(* IEC 61131-3 sources: POC_HINCAPIE/Project/SIEMENS/DIGSI/Guadalupe/TMP/CFC/7344242.46252 (part 2) *)

     (* 0133 - GDL69TRF2F003_.Application.FG1_UserDef.FB2_Universal.SPS6 *)
     EXV_SPS_0133   {COMMENT := "GDL69TRF2F003_.Application.FG1_UserDef.FB2_Universal.SPS6";DESC := "0##Application#Usuario#Logicas#Barra Viva - Linea muerta##1";}:OEXV_BO_SPS;

     (* 0134 - GDL69TRF2F003_.Application.FG1_PowerTransformerStarpoint.FN1_OMV_Fund_1ph.FB1_OpMeas_Fund_1ph_Pres.VxC.CMV_Mag *)
     EXV_MV_0134    {COMMENT := "GDL69TRF2F003_.Application.FG1_PowerTransformerStarpoint.FN1_OMV_Fund_1ph.FB1_OpMeas_Fund_1ph_Pres.VxC.CMV_Mag";DESC := "0##Application#Transform. neut.p 1#Fundamental#Fundam#V#magnitude##1";}:IEXV_MVL_DI;
END_VAR

     EXV_MV_0125         (LNK := 125);

     EXV_MV_0126         (LNK := 126);

     EXV_MV_0127         (LNK := 127);

     EXV_MV_0134         (LNK := 134);

     GT_D_1              (IN1 := EXV_MV_0125.VAL(* POSITION := -1*-1: SIZE := 41* -1:   *) ,
                          IN2 := 80);

     GT_D_2              (IN1 := EXV_MV_0126.VAL(* POSITION := -1*-1: SIZE := 41* -1:   *) ,
                          IN2 := 80);

     GT_D_3              (IN1 := EXV_MV_0127.VAL(* POSITION := -1*-1: SIZE := 41* -1:   *) ,
                          IN2 := 80);

     LT_D_4              (IN1 := EXV_MV_0125.VAL(* POSITION := -1*-1: SIZE := 41* -1:   *) ,
                          IN2 := 110);

     LT_D_5              (IN1 := EXV_MV_0126.VAL(* POSITION := -1*-1: SIZE := 41* -1:   *) ,
                          IN2 := 110);

     LT_D_6              (IN1 := EXV_MV_0127.VAL(* POSITION := -1*-1: SIZE := 41* -1:   *) ,
                          IN2 := 110);

     LT_D_7              (IN1 := EXV_MV_0125.VAL(* POSITION := -1*-1: SIZE := 41* -1:   *) ,
                          IN2 := 40);

     LT_D_8              (IN1 := EXV_MV_0126.VAL(* POSITION := -1*-1: SIZE := 41* -1:   *) ,
                          IN2 := 40);

     LT_D_9              (IN1 := EXV_MV_0127.VAL(* POSITION := -1*-1: SIZE := 41* -1:   *) ,
                          IN2 := 40);

     AND10_10            (X1 := GT_D_1.OUT,
                          X2 := GT_D_2.OUT,
                          X3 := GT_D_3.OUT,
                          X4 := LT_D_4.OUT,
                          X5 := LT_D_5.OUT,
                          X6 := LT_D_6.OUT,
                          X7 := 1,
                          X8 := 1,
                          X9 := 1,
                          X10 := 1);

     LT_D_11             (IN1 := EXV_MV_0134.VAL(* POSITION := -1*-1: SIZE := 38* -1:   *) ,
                          IN2 := 23);

     AND10_12            (X1 := LT_D_7.OUT,
                          X2 := LT_D_8.OUT,
                          X3 := LT_D_9.OUT,
                          X4 := 1,
                          X5 := 1,
                          X6 := 1,
                          X7 := 1,
                          X8 := 1,
                          X9 := 1,
                          X10 := 1);

     AND10_13            (X1 := AND10_10.Y,
                          X2 := LT_D_11.OUT,
                          X3 := 1,
                          X4 := 1,
                          X5 := 1,
                          X6 := 1,
                          X7 := 1,
                          X8 := 1,
                          X9 := 1,
                          X10 := 1);

     AND10_14            (X1 := AND10_12.Y,
                          X2 := LT_D_11.OUT,
                          X3 := 1,
                          X4 := 1,
                          X5 := 1,
                          X6 := 1,
                          X7 := 1,
                          X8 := 1,
                          X9 := 1,
                          X10 := 1);

     OR10_15             (X1 := 0,
                          X2 := AND10_13.Y,
                          X3 := 0,
                          X4 := 0,
                          X5 := 0,
                          X6 := 0,
                          X7 := 0,
                          X8 := 0,
                          X9 := 0,
                          X10 := 0);

     EXV_SPS_0128        (LNK := 128,
                          VAL := AND10_12.Y(* POSITION := -1*-1: SIZE := 27* -1:   *) );
     EXV_SPS_0129        (LNK := 129,
                          VAL := AND10_10.Y(* POSITION := -1*-1: SIZE := 26* -1:   *) );
     EXV_SPS_0130        (LNK := 130,
                          VAL := LT_D_11.OUT(* POSITION := -1*-1: SIZE := 28* -1:   *) );
     EXV_SPS_0131        (LNK := 131,
                          VAL := OR10_15.Y(* POSITION := -1*-1: SIZE := 33* -1:   *) );
     EXV_SPS_0132        (LNK := 132,
                          VAL := AND10_14.Y(* POSITION := -1*-1: SIZE := 35* -1:   *) );
     EXV_SPS_0133        (LNK := 133,
                          VAL := AND10_13.Y(* POSITION := -1*-1: SIZE := 34* -1:   *) );

(* COMMENT_TEXT;{X=65,Y=2};{Width=23, Height=3};FontSize := 10,LineColor := 0,LineWidth := 0,Alignment := Near,AutoWrap := True,BackColor := -16711681,Background := False,TextColor := 0,WallpaperGamma := 100,PartitionID := 1,;Condición de barra muerta *)
(* COMMENT_TEXT;{X=59,Y=28};{Width=22, Height=2};FontSize := 10,LineColor := 0,LineWidth := 0,Alignment := Near,AutoWrap := True,BackColor := -16711681,Background := False,TextColor := 0,WallpaperGamma := 100,PartitionID := 1,;condición de barra viva *)
(* COMMENT_TEXT;{X=182,Y=26};{Width=22, Height=2};FontSize := 10,LineColor := 0,LineWidth := 0,Alignment := Near,AutoWrap := True,BackColor := -16711681,Background := False,TextColor := 0,WallpaperGamma := 100,PartitionID := 1,;Lado 13,8 KV Muerto *)

END_PROGRAM

                                                  (* ---------- Program : CHART_Falla_PTs ----------  *)

PROGRAM CHART_Falla_PTs
{COMMENT := "Falla PTs";DESC := "";}
(* ChartLayout;PageSize := A4,Rows := 3,Columns := 2,MarginMode := WithoutMargins,MarginSize := 37,MarginLines := 1 *)
(* PartitionInfo;Id := 1,Name := Partition_1,Comment :=   *)
VAR

     (* IO_IOVISIBILITY;OR10_1;X3:X4:X5:X6:X7:X8:X9:X10: *)

     (* PartitionInfo;PartitionID OR10_1;1  *)
OR10_1          { COMMENT := 'or10_1'; POSITION := 55,10; SIZE := 12, 12; } :OR10;

     (* IO_IOVISIBILITY;OR10_2;X3:X4:X5:X6:X7:X8:X9:X10: *)

     (* PartitionInfo;PartitionID OR10_2;1  *)
OR10_2          { COMMENT := 'or10_3'; POSITION := 55,23; SIZE := 12, 12; } :OR10;

     (* IO_IOVISIBILITY;AND10_3;X3:X4:X5:X6:X7:X8:X9:X10: *)

     (* PartitionInfo;PartitionID AND10_3;1  *)
AND10_3         { COMMENT := 'and10_1'; POSITION := 74,4; SIZE := 12, 12; } :AND10;

     (* IO_IOVISIBILITY;AND10_4;X4:X5:X6:X7:X8:X9:X10: *)

     (* PartitionInfo;PartitionID AND10_4;1  *)
AND10_4         { COMMENT := 'and10_2'; POSITION := 74,15; SIZE := 12, 12; } :AND10;

     (* IO_IOVISIBILITY;OR10_5;X3:X4:X5:X6:X7:X8:X9:X10: *)

     (* PartitionInfo;PartitionID OR10_5;1  *)
OR10_5          { COMMENT := 'or10_2'; POSITION := 71,41; SIZE := 12, 12; } :OR10;

     (* IO_IOVISIBILITY;OR10_6;X3:X4:X5:X6:X7:X8:X9:X10: *)

     (* PartitionInfo;PartitionID OR10_6;1  *)
OR10_6          { COMMENT := 'or10_4'; POSITION := 105,11; SIZE := 12, 12; } :OR10;

     (* 0135 - GDL69TRF2F003_.Application.FG_PowerSystem.FN1_MUVoltage_3ph.FB1_SMCB.VTmcb *)
     EXV_SPS_0135   {COMMENT := "GDL69TRF2F003_.Application.FG_PowerSystem.FN1_MUVoltage_3ph.FB1_SMCB.VTmcb";DESC := "0##Application#Power system#PTs Barra 69kV#VT miniatureCB#>Open##1";}:OEXV_BO_SPS;

     (* 0136 - GDL69TRF2F003_.Application.FG_PowerSystem.FN1_MUVoltage_1ph.FB1_SMCB.VTmcb *)
     EXV_SPS_0136   {COMMENT := "GDL69TRF2F003_.Application.FG_PowerSystem.FN1_MUVoltage_1ph.FB1_SMCB.VTmcb";DESC := "0##Application#Power system#PTs Barra 13.8kV#VT miniatureCB#>Open##1";}:OEXV_BO_SPS;

     (* 0137 - GDL69TRF2F003_.Application.FG1_UserDef.FB1_Universal.FaPTN3PCyMHV *)
     EXV_SPS_0137   {COMMENT := "GDL69TRF2F003_.Application.FG1_UserDef.FB1_Universal.FaPTN3PCyMHV";DESC := "0##Application#Usuario#Entradas#Falla MCB PT B1_2 69kV PCyM N3##1";}:IEXV_SPS_BO;

     (* 0138 - GDL69TRF2F003_.Application.FG1_UserDef.FB2_Universal.FaPTAlta *)
     EXV_SPS_0138   {COMMENT := "GDL69TRF2F003_.Application.FG1_UserDef.FB2_Universal.FaPTAlta";DESC := "0##Application#Usuario#Logicas#Falla PT Alta##1";}:OEXV_BO_SPS;

     (* 0139 - GDL69TRF2F003_.Application.FG1_UserDef.FB2_Universal.FaPTBaja *)
     EXV_SPS_0139   {COMMENT := "GDL69TRF2F003_.Application.FG1_UserDef.FB2_Universal.FaPTBaja";DESC := "0##Application#Usuario#Logicas#Falla PT Baja##1";}:OEXV_BO_SPS;

     (* 0140 - GDL69TRF2F003_.Application.FG1_UserDef.FB1_Universal.FaPTN2PCyMLV *)
     EXV_SPS_0140   {COMMENT := "GDL69TRF2F003_.Application.FG1_UserDef.FB1_Universal.FaPTN2PCyMLV";DESC := "0##Application#Usuario#Entradas#Falla MCB PT 13.8kV PCyM N3##1";}:IEXV_SPS_BO;

     (* 0141 - GDL69TRF2F003_.Application.FG1_UserDef.FB1_Universal.FaPTN2TUJLV *)
     EXV_SPS_0141   {COMMENT := "GDL69TRF2F003_.Application.FG1_UserDef.FB1_Universal.FaPTN2TUJLV";DESC := "0##Application#Usuario#Entradas#Falla MCB PT 13.8kV 9TUJ N3##1";}:IEXV_SPS_BO;

     (* 0142 - GDL69TRF2F003_.Application.FG1_UserDef.FB1_Universal.SPS3 *)
     EXV_SPS_0142   {COMMENT := "GDL69TRF2F003_.Application.FG1_UserDef.FB1_Universal.SPS3";DESC := "0##Application#Usuario#Entradas#Posicion Q2 Cerrado##1";}:IEXV_SPS_BO;

     (* 0143 - GDL69TRF2F003_.Application.FG1_UserDef.FB3_Universal.RxPosQ1.DPC_StatusOn *)
     EXV_SPS_0143   {COMMENT := "GDL69TRF2F003_.Application.FG1_UserDef.FB3_Universal.RxPosQ1.DPC_StatusOn";DESC := "0##Application#Usuario#Rx Goose#Posicion 6T4-Q1#closed##1";}:IEXV_SPS_BO;

     (* 0144 - GDL69TRF2F003_.Application.FG1_UserDef.FB1_Universal.FaPTN3Bar1HV *)
     EXV_SPS_0144   {COMMENT := "GDL69TRF2F003_.Application.FG1_UserDef.FB1_Universal.FaPTN3Bar1HV";DESC := "0##Application#Usuario#Entradas#Falla MCB PT B1 69kV 6TUJ1 N3##1";}:IEXV_SPS_BO;

     (* 0145 - GDL69TRF2F003_.Application.FG1_UserDef.FB1_Universal.FaPTN3Bar2HV *)
     EXV_SPS_0145   {COMMENT := "GDL69TRF2F003_.Application.FG1_UserDef.FB1_Universal.FaPTN3Bar2HV";DESC := "0##Application#Usuario#Entradas#Falla MCB PT B2 69kV 6TUJ2 N3##1";}:IEXV_SPS_BO;
END_VAR

     EXV_SPS_0137        (LNK := 137);

     EXV_SPS_0140        (LNK := 140);

     EXV_SPS_0141        (LNK := 141);

     EXV_SPS_0142        (LNK := 142);

     EXV_SPS_0143        (LNK := 143);

     EXV_SPS_0144        (LNK := 144);

     EXV_SPS_0145        (LNK := 145);

     OR10_1              (X1 := EXV_SPS_0137.VAL(* POSITION := 14*13: SIZE := 37* -1:   *) ,
                          X2 := EXV_SPS_0145.VAL(* POSITION := 15*14: SIZE := 36* -1:   *) ,
                          X3 := 0,
                          X4 := 0,
                          X5 := 0,
                          X6 := 0,
                          X7 := 0,
                          X8 := 0,
                          X9 := 0,
                          X10 := 0);

     OR10_2              (X1 := EXV_SPS_0137.VAL(* POSITION := 12*26: SIZE := 37* -1:   *) ,
                          X2 := EXV_SPS_0144.VAL(* POSITION := -1*-1: SIZE := 36* -1:   *) ,
                          X3 := 0,
                          X4 := 0,
                          X5 := 0,
                          X6 := 0,
                          X7 := 0,
                          X8 := 0,
                          X9 := 0,
                          X10 := 0);

     AND10_3             (X1 := EXV_SPS_0142.VAL(* POSITION := -1*-1: SIZE := 31* -1:   *) ,
                          X2 := OR10_1.Y,
                          X3 := 1,
                          X4 := 1,
                          X5 := 1,
                          X6 := 1,
                          X7 := 1,
                          X8 := 1,
                          X9 := 1,
                          X10 := 1);

     AND10_4             (X1 := EXV_SPS_0143.VAL(* POSITION := -1*-1: SIZE := 33* -1:   *) ,
                          X2 := NOT EXV_SPS_0142.VAL(* POSITION := -1*-1: SIZE := 31* -1:   *) ,
                          X3 := OR10_2.Y,
                          X4 := 1,
                          X5 := 1,
                          X6 := 1,
                          X7 := 1,
                          X8 := 1,
                          X9 := 1,
                          X10 := 1);

     OR10_5              (X1 := EXV_SPS_0140.VAL(* POSITION := -1*-1: SIZE := 35* -1:   *) ,
                          X2 := EXV_SPS_0141.VAL(* POSITION := -1*-1: SIZE := 35* -1:   *) ,
                          X3 := 0,
                          X4 := 0,
                          X5 := 0,
                          X6 := 0,
                          X7 := 0,
                          X8 := 0,
                          X9 := 0,
                          X10 := 0);

     OR10_6              (X1 := AND10_3.Y,
                          X2 := AND10_4.Y,
                          X3 := 0,
                          X4 := 0,
                          X5 := 0,
                          X6 := 0,
                          X7 := 0,
                          X8 := 0,
                          X9 := 0,
                          X10 := 0);

     EXV_SPS_0135        (LNK := 135,
                          VAL := OR10_6.Y(* POSITION := -1*-1: SIZE := 37* -1:   *) );
     EXV_SPS_0136        (LNK := 136,
                          VAL := OR10_5.Y(* POSITION := 90*45: SIZE := 38* -1:   *) );
     EXV_SPS_0138        (LNK := 138,
                          VAL := OR10_6.Y(* POSITION := -1*-1: SIZE := 28* -1:   *) );
     EXV_SPS_0139        (LNK := 139,
                          VAL := OR10_5.Y(* POSITION := 90*44: SIZE := 28* -1:   *) );

(* COMMENT_TEXT;{X=17,Y=39};{Width=17, Height=1};FontSize := 10,LineColor := 0,LineWidth := 0,Alignment := Near,AutoWrap := True,BackColor := -16711681,Background := False,TextColor := 0,WallpaperGamma := 100,PartitionID := 1,;Falla Mcb PT lado 13.8 kV *)
(* COMMENT_TEXT;{X=16,Y=3};{Width=17, Height=1};FontSize := 10,LineColor := 0,LineWidth := 0,Alignment := Near,AutoWrap := True,BackColor := -16711681,Background := False,TextColor := 0,WallpaperGamma := 100,PartitionID := 1,;Falla Mcb PT lado 69 kV *)
(* COMMENT_TEXT;{X=8,Y=18};{Width=17, Height=1};FontSize := 10,LineColor := 0,LineWidth := 0,Alignment := Near,AutoWrap := True,BackColor := -256,Background := False,TextColor := 0,WallpaperGamma := 100,PartitionID := 1,;GOOSE Pos Q1 F002 *)

END_PROGRAM

                                                  (* ---------- Program : CHART_Interlocking ----------  *)

PROGRAM CHART_Interlocking
{COMMENT := "Interlocking";DESC := "";}
(* ChartLayout;PageSize := A4,Rows := 3,Columns := 2,MarginMode := WithoutMargins,MarginSize := 37,MarginLines := 1 *)
(* PartitionInfo;Id := 1,Name := Partition_1,Comment :=    *)
VAR

     (* IO_IOVISIBILITY;AND10_1;X5:X6:X7:X8:X9:X10: *)

     (* PartitionInfo;PartitionID AND10_1;1  *)
AND10_1         { COMMENT := 'and10_4'; POSITION := 68,2; SIZE := 12, 12; } :AND10;

     (* IO_IOVISIBILITY;AND10_2;X5:X6:X7:X8:X9:X10: *)

     (* PartitionInfo;PartitionID AND10_2;1  *)
AND10_2         { COMMENT := 'and10_5'; POSITION := 68,12; SIZE := 12, 12; } :AND10;

     (* IO_IOVISIBILITY;OR10_3;X3:X4:X5:X6:X7:X8:X9:X10: *)

     (* PartitionInfo;PartitionID OR10_3;1  *)
OR10_3          { COMMENT := 'or10_1'; POSITION := 87,7; SIZE := 12, 12; } :OR10;

     (* IO_IOVISIBILITY;AND10_4;X6:X7:X8:X9:X10: *)

     (* PartitionInfo;PartitionID AND10_4;1  *)
AND10_4         { COMMENT := 'and10_1'; POSITION := 67,26; SIZE := 12, 12; } :AND10;

     (* IO_IOVISIBILITY;AND10_5;X5:X6:X7:X8:X9:X10: *)

     (* PartitionInfo;PartitionID AND10_5;1  *)
AND10_5         { COMMENT := 'and10_3'; POSITION := 67,38; SIZE := 12, 12; } :AND10;

     (* IO_IOVISIBILITY;AND10_6;X3:X4:X5:X6:X7:X8:X9:X10: *)

     (* PartitionInfo;PartitionID AND10_6;1  *)
AND10_6         { COMMENT := 'and10_2'; POSITION := 92,32; SIZE := 12, 12; } :AND10;

     (* 0146 - GDL69TRF2F003_.Application.FG_PowerSystem.FN1_MUVoltage_1ph.FB1_SMCB.VTmcb *)
     EXV_SPS_0146   {COMMENT := "GDL69TRF2F003_.Application.FG_PowerSystem.FN1_MUVoltage_1ph.FB1_SMCB.VTmcb";DESC := "0##Application#Power system#PTs Barra 13.8kV#VT miniatureCB#>Open##1";}:IEXV_SPS_BO;

     (* 0147 - GDL69TRF2F003_.Application.FG1_UserDef.FB2_Universal.SPS10 *)
     EXV_SPS_0147   {COMMENT := "GDL69TRF2F003_.Application.FG1_UserDef.FB2_Universal.SPS10";DESC := "0##Application#Usuario#Logicas#Condicion de Sincronismo##1";}:IEXV_SPS_BO;

     (* 0148 - GDL69TRF2F003_.Application.FG1_Breaker_3pol.FB1_CILO.EnaClsFix *)
     EXV_SPS_0148   {COMMENT := "GDL69TRF2F003_.Application.FG1_Breaker_3pol.FB1_CILO.EnaClsFix";DESC := "0##Application#Interruptor HV#Interlocking#>Enable closing (fixed)##1";}:OEXV_BO_SPS;

     (* 0149 - GDL69TRF2F003_.Application.FG1_UserDef.FB2_Universal.SPS14 *)
     EXV_SPS_0149   {COMMENT := "GDL69TRF2F003_.Application.FG1_UserDef.FB2_Universal.SPS14";DESC := "0##Application#Usuario#Logicas#Permisivo Q0 CLS 1 Display##1";}:OEXV_BO_SPS;

     (* 0150 - GDL69TRF2F003_.Application.FG1_UserDef.FB2_Universal.SPS15 *)
     EXV_SPS_0150   {COMMENT := "GDL69TRF2F003_.Application.FG1_UserDef.FB2_Universal.SPS15";DESC := "0##Application#Usuario#Logicas#Permisivo Q0 CLS 2 Display##1";}:OEXV_BO_SPS;

     (* 0151 - GDL69TRF2F003_.Application.FG1_UserDef.FB1_Universal.SPS2 *)
     EXV_SPS_0151   {COMMENT := "GDL69TRF2F003_.Application.FG1_UserDef.FB1_Universal.SPS2";DESC := "0##Application#Usuario#Entradas#Posicion Int Q0 Cerrado##1";}:IEXV_SPS_BO;

     (* 0152 - GDL69TRF2F003_.Application.FG1_UserDef.FB1_Universal.Op86T *)
     EXV_SPS_0152   {COMMENT := "GDL69TRF2F003_.Application.FG1_UserDef.FB1_Universal.Op86T";DESC := "0##Application#Usuario#Entradas#Opero 86T##1";}:IEXV_SPS_BO;

     (* 0153 - GDL69TRF2F003_.Application.FG1_UserDef.FB3_Universal.RxPosQ013.DPC_StatusOn *)
     EXV_SPS_0153   {COMMENT := "GDL69TRF2F003_.Application.FG1_UserDef.FB3_Universal.RxPosQ013.DPC_StatusOn";DESC := "0##Application#Usuario#Rx Goose#Posicion 9T6-Q0#closed##1";}:IEXV_SPS_BO;

     (* 0154 - GDL69TRF2F003_.Application.FG1_UserDef.FB3_Universal.Rx86BFB169 *)
     EXV_SPS_0154   {COMMENT := "GDL69TRF2F003_.Application.FG1_UserDef.FB3_Universal.Rx86BFB169";DESC := "0##Application#Usuario#Rx Goose#Opero 86BF B1 69 kV##1";}:IEXV_SPS_BO;

     (* 0155 - GDL69TRF2F003_.Application.FG1_UserDef.FB3_Universal.Rx86BFB269 *)
     EXV_SPS_0155   {COMMENT := "GDL69TRF2F003_.Application.FG1_UserDef.FB3_Universal.Rx86BFB269";DESC := "0##Application#Usuario#Rx Goose#Opero 86BF B2 69 kV##1";}:IEXV_SPS_BO;

     (* 0156 - GDL69TRF2F003_.Application.FG1_UserDef.FB3_Universal.Rx86BF13 *)
     EXV_SPS_0156   {COMMENT := "GDL69TRF2F003_.Application.FG1_UserDef.FB3_Universal.Rx86BF13";DESC := "0##Application#Usuario#Rx Goose#Opero 86BF 13.8 kV##1";}:IEXV_SPS_BO;

     (* 0157 - GDL69TRF2F003_.Application.FG1_UserDef.FB2_Universal.SPS *)
     EXV_SPS_0157   {COMMENT := "GDL69TRF2F003_.Application.FG1_UserDef.FB2_Universal.SPS";DESC := "0##Application#Usuario#Logicas#Condicion B1 OK##1";}:OEXV_BO_SPS;

     (* 0158 - GDL69TRF2F003_.Application.FG1_UserDef.FB2_Universal.SPS1 *)
     EXV_SPS_0158   {COMMENT := "GDL69TRF2F003_.Application.FG1_UserDef.FB2_Universal.SPS1";DESC := "0##Application#Usuario#Logicas#Condicion B2 OK##1";}:OEXV_BO_SPS;

     (* 0159 - GDL69TRF2F003_.Application.FG1_UserDef.FB2_Universal.SPS2 *)
     EXV_SPS_0159   {COMMENT := "GDL69TRF2F003_.Application.FG1_UserDef.FB2_Universal.SPS2";DESC := "0##Application#Usuario#Logicas#Condicion B1/B2 OK##1";}:OEXV_BO_SPS;

     (* 0160 - GDL69TRF2F003_.Application.FG1_UserDef.FB3_Universal.RxPosQ1.DPC_StatusOn *)
     EXV_SPS_0160   {COMMENT := "GDL69TRF2F003_.Application.FG1_UserDef.FB3_Universal.RxPosQ1.DPC_StatusOn";DESC := "0##Application#Usuario#Rx Goose#Posicion 6T4-Q1#closed##1";}:IEXV_SPS_BO;

     (* 0161 - GDL69TRF2F003_.Application.FG1_UserDef.FB1_Universal.SPS3 *)
     EXV_SPS_0161   {COMMENT := "GDL69TRF2F003_.Application.FG1_UserDef.FB1_Universal.SPS3";DESC := "0##Application#Usuario#Entradas#Posicion Q2 Cerrado##1";}:IEXV_SPS_BO;

     (* 0162 - GDL69TRF2F003_.Application.FG1_UserDef.FB1_Universal.FaPTN3PCyMHV *)
     EXV_SPS_0162   {COMMENT := "GDL69TRF2F003_.Application.FG1_UserDef.FB1_Universal.FaPTN3PCyMHV";DESC := "0##Application#Usuario#Entradas#Falla MCB PT B1_2 69kV PCyM N3##1";}:IEXV_SPS_BO;

     (* 0163 - GDL69TRF2F003_.Application.FG1_UserDef.FB1_Universal.FaPTN3Bar1HV *)
     EXV_SPS_0163   {COMMENT := "GDL69TRF2F003_.Application.FG1_UserDef.FB1_Universal.FaPTN3Bar1HV";DESC := "0##Application#Usuario#Entradas#Falla MCB PT B1 69kV 6TUJ1 N3##1";}:IEXV_SPS_BO;

     (* 0164 - GDL69TRF2F003_.Application.FG1_UserDef.FB1_Universal.FaPTN3Bar2HV *)
     EXV_SPS_0164   {COMMENT := "GDL69TRF2F003_.Application.FG1_UserDef.FB1_Universal.FaPTN3Bar2HV";DESC := "0##Application#Usuario#Entradas#Falla MCB PT B2 69kV 6TUJ2 N3##1";}:IEXV_SPS_BO;

     (* 0165 - GDL69TRF2F003_.Application.FG1_UserDef.FB2_Universal.SCDB2 *)
     EXV_SPS_0165   {COMMENT := "GDL69TRF2F003_.Application.FG1_UserDef.FB2_Universal.SCDB2";DESC := "0##Application#Usuario#Logicas#Falla SBD2##1";}:IEXV_SPS_BO;

     (* 0166 - GDL69TRF2F003_.Application.FG1_UserDef.FB3_Universal.RxAnormBCU *)
     EXV_SPS_0166   {COMMENT := "GDL69TRF2F003_.Application.FG1_UserDef.FB3_Universal.RxAnormBCU";DESC := "0##Application#Usuario#Rx Goose#Anormalidad BCU##1";}:IEXV_SPS_BO;
END_VAR

     EXV_SPS_0146        (LNK := 146);

     EXV_SPS_0147        (LNK := 147);

     EXV_SPS_0151        (LNK := 151);

     EXV_SPS_0152        (LNK := 152);

     EXV_SPS_0153        (LNK := 153);

     EXV_SPS_0154        (LNK := 154);

     EXV_SPS_0155        (LNK := 155);

     EXV_SPS_0156        (LNK := 156);

     EXV_SPS_0160        (LNK := 160);

     EXV_SPS_0161        (LNK := 161);

     EXV_SPS_0162        (LNK := 162);

     EXV_SPS_0163        (LNK := 163);

     EXV_SPS_0164        (LNK := 164);

     EXV_SPS_0165        (LNK := 165);

     EXV_SPS_0166        (LNK := 166);

     AND10_1             (X1 := EXV_SPS_0160.VAL(* POSITION := 28*5: SIZE := 33* -1:   *) ,
                          X2 := NOT EXV_SPS_0154.VAL(* POSITION := 30*6: SIZE := 31* -1:   *) ,
                          X3 := NOT EXV_SPS_0162.VAL(* POSITION := 24*7: SIZE := 37* -1:   *) ,
                          X4 := NOT EXV_SPS_0163.VAL(* POSITION := 25*8: SIZE := 36* -1:   *) ,
                          X5 := 1,
                          X6 := 1,
                          X7 := 1,
                          X8 := 1,
                          X9 := 1,
                          X10 := 1);

     AND10_2             (X1 := EXV_SPS_0161.VAL(* POSITION := 29*15: SIZE := 31* -1:   *) ,
                          X2 := NOT EXV_SPS_0155.VAL(* POSITION := 29*16: SIZE := 31* -1:   *) ,
                          X3 := NOT EXV_SPS_0162.VAL(* POSITION := 23*17: SIZE := 37* -1:   *) ,
                          X4 := NOT EXV_SPS_0164.VAL(* POSITION := 24*18: SIZE := 36* -1:   *) ,
                          X5 := 1,
                          X6 := 1,
                          X7 := 1,
                          X8 := 1,
                          X9 := 1,
                          X10 := 1);

     OR10_3              (X1 := AND10_1.Y,
                          X2 := AND10_2.Y,
                          X3 := 0,
                          X4 := 0,
                          X5 := 0,
                          X6 := 0,
                          X7 := 0,
                          X8 := 0,
                          X9 := 0,
                          X10 := 0);

     AND10_4             (X1 := OR10_3.Y,
                          X2 := NOT EXV_SPS_0151.VAL(* POSITION := 27*30: SIZE := 33* -1:   *) ,
                          X3 := NOT EXV_SPS_0153.VAL(* POSITION := 27*31: SIZE := 33* -1:   *) ,
                          X4 := NOT EXV_SPS_0152.VAL(* POSITION := 34*32: SIZE := 26* -1:   *) ,
                          X5 := NOT EXV_SPS_0156.VAL(* POSITION := 29*33: SIZE := 31* -1:   *) ,
                          X6 := 1,
                          X7 := 1,
                          X8 := 1,
                          X9 := 1,
                          X10 := 1);

     AND10_5             (X1 := NOT EXV_SPS_0165.VAL(* POSITION := 34*41: SIZE := 26* -1:   *) ,
                          X2 := NOT EXV_SPS_0146.VAL(* POSITION := 22*42: SIZE := 38* -1:   *) ,
                          X3 := EXV_SPS_0166.VAL(* POSITION := -1*-1: SIZE := 29* -1:   *) ,
                          X4 := EXV_SPS_0147.VAL(* POSITION := 27*44: SIZE := 33* -1:   *) ,
                          X5 := 1,
                          X6 := 1,
                          X7 := 1,
                          X8 := 1,
                          X9 := 1,
                          X10 := 1);

     AND10_6             (X1 := AND10_4.Y,
                          X2 := AND10_5.Y,
                          X3 := 1,
                          X4 := 1,
                          X5 := 1,
                          X6 := 1,
                          X7 := 1,
                          X8 := 1,
                          X9 := 1,
                          X10 := 1);

     EXV_SPS_0148        (LNK := 148,
                          VAL := AND10_6.Y(* POSITION := 111*35: SIZE := 39* -1:   *) );
     EXV_SPS_0149        (LNK := 149,
                          VAL := AND10_4.Y(* POSITION := 83*24: SIZE := 34* -1:   *) );
     EXV_SPS_0150        (LNK := 150,
                          VAL := AND10_5.Y(* POSITION := 86*41: SIZE := 34* -1:   *) );
     EXV_SPS_0157        (LNK := 157,
                          VAL := AND10_1.Y(* POSITION := 88*5: SIZE := 29* -1:   *) );
     EXV_SPS_0158        (LNK := 158,
                          VAL := AND10_2.Y(* POSITION := 87*15: SIZE := 29* -1:   *) );
     EXV_SPS_0159        (LNK := 159,
                          VAL := OR10_3.Y(* POSITION := 107*9: SIZE := 30* -1:   *) );

(* COMMENT_TEXT;{X=3,Y=6};{Width=18, Height=1};FontSize := 8,LineColor := 0,LineWidth := 0,Alignment := Near,AutoWrap := True,BackColor := -256,Background := False,TextColor := 0,WallpaperGamma := 100,PartitionID := 1,;GOOSE 86BF B1 69kV No Op BCU *)
(* COMMENT_TEXT;{X=6,Y=31};{Width=14, Height=1};FontSize := 8,LineColor := 0,LineWidth := 0,Alignment := Near,AutoWrap := True,BackColor := -256,Background := False,TextColor := 0,WallpaperGamma := 100,PartitionID := 1,;GOOSE Pos 9T6-Q0 F004 *)
(* COMMENT_TEXT;{X=6,Y=33};{Width=19, Height=1};FontSize := 8,LineColor := 0,LineWidth := 0,Alignment := Near,AutoWrap := True,BackColor := -256,Background := False,TextColor := 0,WallpaperGamma := 100,PartitionID := 1,;GOOSE 86BF 13.8kV No Op F004 *)
(* COMMENT_TEXT;{X=3,Y=16};{Width=18, Height=1};FontSize := 8,LineColor := 0,LineWidth := 0,Alignment := Near,AutoWrap := True,BackColor := -256,Background := False,TextColor := 0,WallpaperGamma := 100,PartitionID := 1,;GOOSE 86BF B2 69kV No Op BCU *)
(* COMMENT_TEXT;{X=3,Y=5};{Width=18, Height=1};FontSize := 8,LineColor := 0,LineWidth := 0,Alignment := Near,AutoWrap := True,BackColor := -256,Background := False,TextColor := 0,WallpaperGamma := 100,PartitionID := 1,;GOOSE Pos Q1 F002 *)
(* COMMENT_TEXT;{X=7,Y=43};{Width=13, Height=1};FontSize := 8,LineColor := 0,LineWidth := 0,Alignment := Near,AutoWrap := True,BackColor := -256,Background := False,TextColor := 0,WallpaperGamma := 100,PartitionID := 1,;GOOSE Anorm BCU F002 *)

END_PROGRAM

CONFIGURATION  PLC_CONTROL
   RESOURCE PLANS { COMMENT := "Txt100_100";} ON CPU32
     TASK EVENT_SLOW     { TICKS := 1300;}(PRIORITY := INTERNAL);
     TASK EVENT_FAST     { TICKS := 255;}(PRIORITY := INTERNAL);
     TASK MEASUREMENT    { TICKS := 2536;}(PRIORITY := INTERNAL);
     TASK INTERLOCKING   { TICKS := 2173;}(PRIORITY := INTERNAL);

     PROGRAM FBI001 WITH EVENT_SLOW:  CHART_Alarmas;
     PROGRAM FBI002 WITH EVENT_FAST:  CHART_Arranque_50BF;
     PROGRAM FBI003 WITH EVENT_SLOW:  CHART_Disparo_por_Fases;
     PROGRAM FBI004 WITH EVENT_SLOW:  CHART_Falla_Goose;
     PROGRAM FBI005 WITH EVENT_SLOW:  CHART_Posiciones;
     PROGRAM FBI006 WITH EVENT_SLOW:  CHART_Synchrocheck;
     PROGRAM FBI007 WITH EVENT_SLOW:  CHART_Sincronismo;
     PROGRAM FBI008 WITH EVENT_SLOW:  CHART_Falla_PTs;
     PROGRAM FBI009 WITH EVENT_SLOW:  CHART_Interlocking;

   END_RESOURCE

 END_CONFIGURATION
